// TIA Portal V20 export
FUNCTION_BLOCK "Simulation"   // FB193, LAD
// stored: MemoryReserve 100, Namespace Unit1.Em4, SetENOAutomatically false
   VAR_INPUT
      simulation { ExternalAccessible := 'False'; ExternalVisible := 'False'; ExternalWritable := 'False'} : Bool;
   END_VAR
   VAR
      instActuator { ExternalAccessible := 'False'; ExternalVisible := 'False'; ExternalWritable := 'False'} : Array[0..19] of "Simulation_Actuator";
      statDigitalSignal { ExternalAccessible := 'False'; ExternalVisible := 'False'; ExternalWritable := 'False'} : Array[0..9] of Bool;
   END_VAR
   VAR_TEMP
      tempTRPnPleftPlace : Bool;
   END_VAR
   VAR_TEMP   // added for the SCL form of the ladder/FBD networks
      _w1 : Bool;
   END_VAR
BEGIN

REGION Network 1: Digital Signal
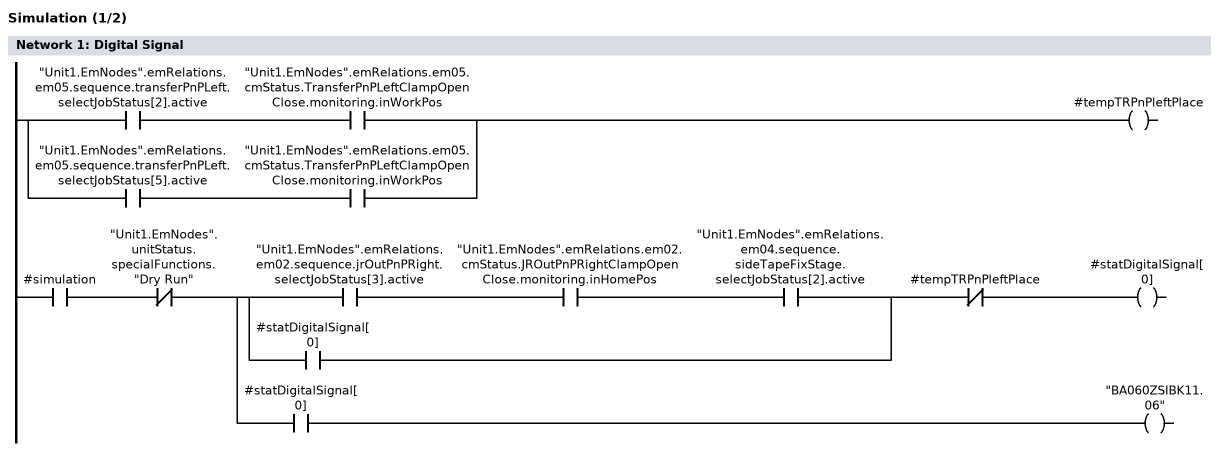
   RUNG wire#powerrail
      Contact( "Unit1.EmNodes".emRelations.em05.sequence.transferPnPLeft.selectJobStatus[2].active )
      Contact( "Unit1.EmNodes".emRelations.em05.cmStatus.TransferPnPLeftClampOpenClose.monitoring.inWorkPos )
      wire#w1
      Coil( #tempTRPnPleftPlace )
   END_RUNG
   RUNG wire#powerrail
      Contact( "Unit1.EmNodes".emRelations.em05.sequence.transferPnPLeft.selectJobStatus[5].active )
      Contact( "Unit1.EmNodes".emRelations.em05.cmStatus.TransferPnPLeftClampOpenClose.monitoring.inWorkPos )
   END_RUNG wire#w1
   RUNG wire#powerrail
      Contact( #simulation )
      I_Contact( "Unit1.EmNodes".unitStatus.specialFunctions."Dry Run" )
      wire#w2
      Contact( "Unit1.EmNodes".emRelations.em02.sequence.jrOutPnPRight.selectJobStatus[3].active )
      Contact( "Unit1.EmNodes".emRelations.em02.cmStatus.JROutPnPRightClampOpenClose.monitoring.inHomePos )
      Contact( "Unit1.EmNodes".emRelations.em04.sequence.sideTapeFixStage.selectJobStatus[2].active )
      wire#w3
      I_Contact( #tempTRPnPleftPlace )
      Coil( #statDigitalSignal[0] )
   END_RUNG
   RUNG wire#w2
      Contact( #statDigitalSignal[0] )
   END_RUNG wire#w3
   RUNG wire#w2
      Contact( #statDigitalSignal[0] )
      Coil( "BA060ZSIBK11.06" )
   END_RUNG
   // the same network as SCL:
   #tempTRPnPleftPlace := ("Unit1.EmNodes".emRelations.em05.sequence.transferPnPLeft.selectJobStatus[2].active AND "Unit1.EmNodes".emRelations.em05.cmStatus.TransferPnPLeftClampOpenClose.monitoring.inWorkPos) OR ("Unit1.EmNodes".emRelations.em05.sequence.transferPnPLeft.selectJobStatus[5].active AND "Unit1.EmNodes".emRelations.em05.cmStatus.TransferPnPLeftClampOpenClose.monitoring.inWorkPos);
   #_w1 := #simulation AND NOT "Unit1.EmNodes".unitStatus.specialFunctions."Dry Run";
   #statDigitalSignal[0] := #_w1 AND (("Unit1.EmNodes".emRelations.em02.sequence.jrOutPnPRight.selectJobStatus[3].active AND "Unit1.EmNodes".emRelations.em02.cmStatus.JROutPnPRightClampOpenClose.monitoring.inHomePos AND "Unit1.EmNodes".emRelations.em04.sequence.sideTapeFixStage.selectJobStatus[2].active) OR #statDigitalSignal[0]) AND NOT #tempTRPnPleftPlace;
   "BA060ZSIBK11.06" := #_w1 AND #statDigitalSignal[0];
END_REGION

REGION Network 2: Two Way Actuator
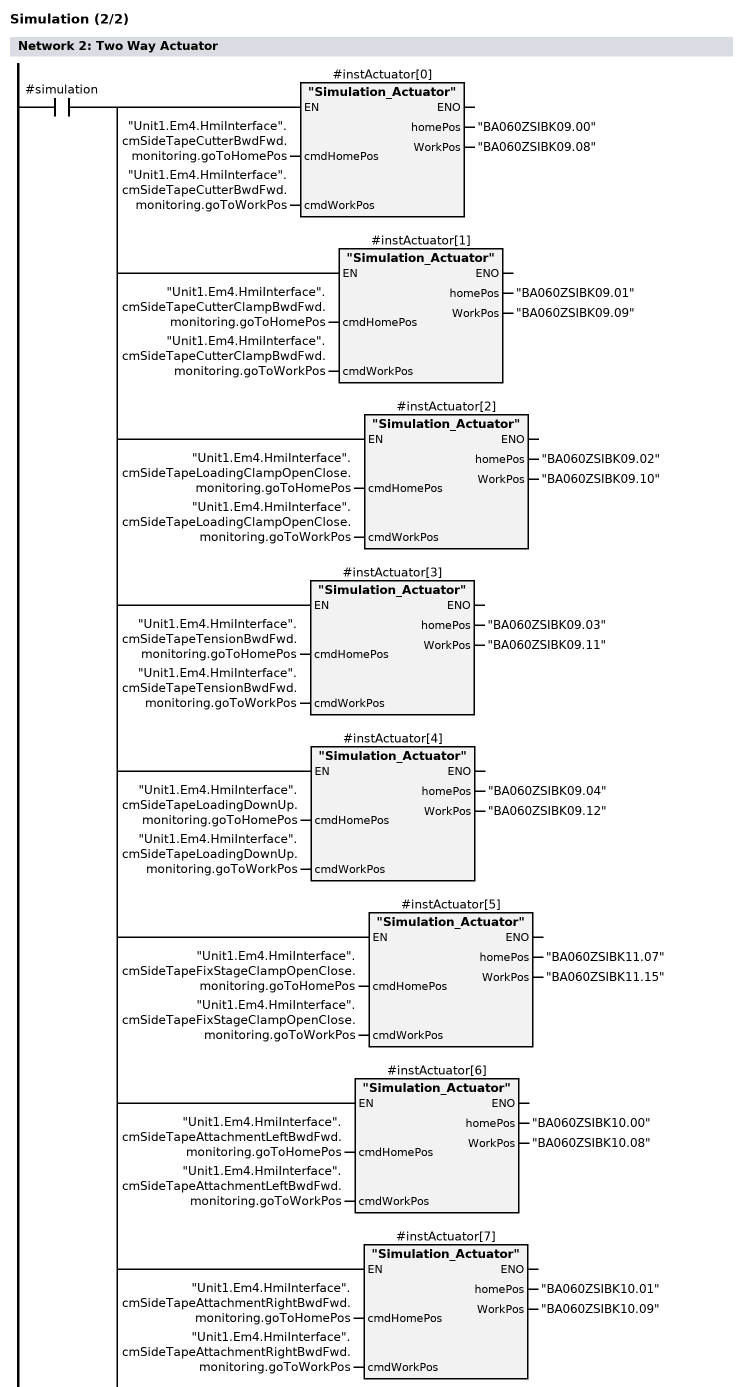
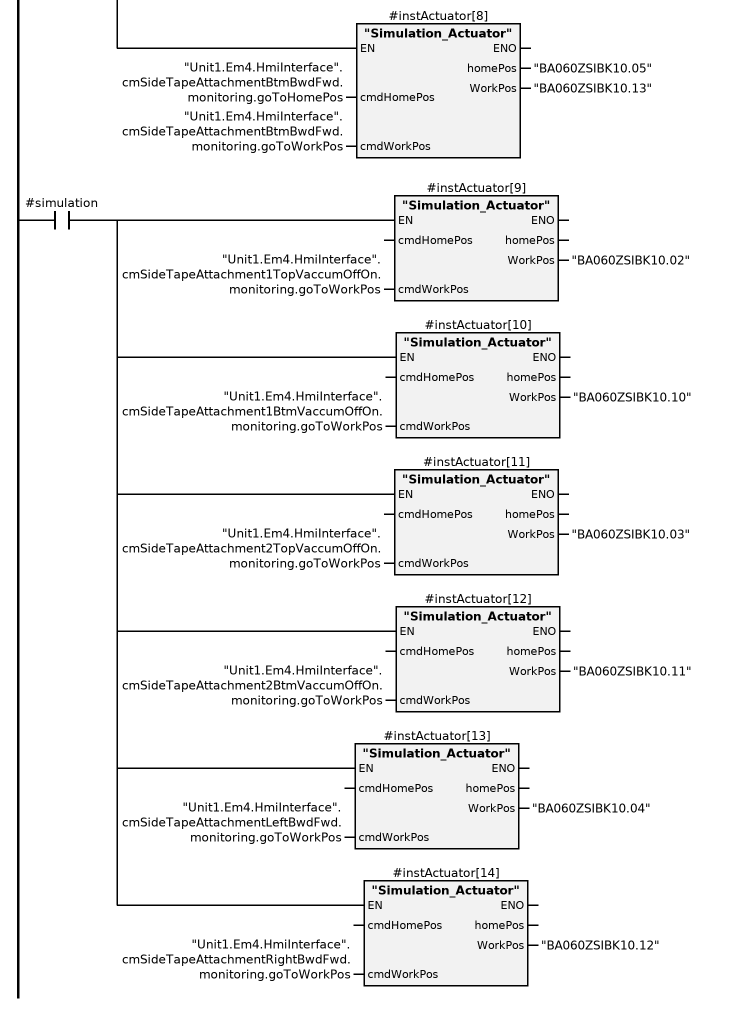
   RUNG wire#powerrail
      Contact( #simulation )
      wire#w1
      #instActuator[0](cmdHomePos := "Unit1.Em4.HmiInterface".cmSideTapeCutterBwdFwd.monitoring.goToHomePos, cmdWorkPos := "Unit1.Em4.HmiInterface".cmSideTapeCutterBwdFwd.monitoring.goToWorkPos, homePos => "BA060ZSIBK09.00", WorkPos => "BA060ZSIBK09.08")
   END_RUNG
   RUNG wire#w1
      #instActuator[1](cmdHomePos := "Unit1.Em4.HmiInterface".cmSideTapeCutterClampBwdFwd.monitoring.goToHomePos, cmdWorkPos := "Unit1.Em4.HmiInterface".cmSideTapeCutterClampBwdFwd.monitoring.goToWorkPos, homePos => "BA060ZSIBK09.01", WorkPos => "BA060ZSIBK09.09")
   END_RUNG
   RUNG wire#w1
      #instActuator[2](cmdHomePos := "Unit1.Em4.HmiInterface".cmSideTapeLoadingClampOpenClose.monitoring.goToHomePos, cmdWorkPos := "Unit1.Em4.HmiInterface".cmSideTapeLoadingClampOpenClose.monitoring.goToWorkPos, homePos => "BA060ZSIBK09.02", WorkPos => "BA060ZSIBK09.10")
   END_RUNG
   RUNG wire#w1
      #instActuator[3](cmdHomePos := "Unit1.Em4.HmiInterface".cmSideTapeTensionBwdFwd.monitoring.goToHomePos, cmdWorkPos := "Unit1.Em4.HmiInterface".cmSideTapeTensionBwdFwd.monitoring.goToWorkPos, homePos => "BA060ZSIBK09.03", WorkPos => "BA060ZSIBK09.11")
   END_RUNG
   RUNG wire#w1
      #instActuator[4](cmdHomePos := "Unit1.Em4.HmiInterface".cmSideTapeLoadingDownUp.monitoring.goToHomePos, cmdWorkPos := "Unit1.Em4.HmiInterface".cmSideTapeLoadingDownUp.monitoring.goToWorkPos, homePos => "BA060ZSIBK09.04", WorkPos => "BA060ZSIBK09.12")
   END_RUNG
   RUNG wire#w1
      #instActuator[5](cmdHomePos := "Unit1.Em4.HmiInterface".cmSideTapeFixStageClampOpenClose.monitoring.goToHomePos, cmdWorkPos := "Unit1.Em4.HmiInterface".cmSideTapeFixStageClampOpenClose.monitoring.goToWorkPos, homePos => "BA060ZSIBK11.07", WorkPos => "BA060ZSIBK11.15")
   END_RUNG
   RUNG wire#w1
      #instActuator[6](cmdHomePos := "Unit1.Em4.HmiInterface".cmSideTapeAttachmentLeftBwdFwd.monitoring.goToHomePos, cmdWorkPos := "Unit1.Em4.HmiInterface".cmSideTapeAttachmentLeftBwdFwd.monitoring.goToWorkPos, homePos => "BA060ZSIBK10.00", WorkPos => "BA060ZSIBK10.08")
   END_RUNG
   RUNG wire#w1
      #instActuator[7](cmdHomePos := "Unit1.Em4.HmiInterface".cmSideTapeAttachmentRightBwdFwd.monitoring.goToHomePos, cmdWorkPos := "Unit1.Em4.HmiInterface".cmSideTapeAttachmentRightBwdFwd.monitoring.goToWorkPos, homePos => "BA060ZSIBK10.01", WorkPos => "BA060ZSIBK10.09")
   END_RUNG
   RUNG wire#w1
      #instActuator[8](cmdHomePos := "Unit1.Em4.HmiInterface".cmSideTapeAttachmentBtmBwdFwd.monitoring.goToHomePos, cmdWorkPos := "Unit1.Em4.HmiInterface".cmSideTapeAttachmentBtmBwdFwd.monitoring.goToWorkPos, homePos => "BA060ZSIBK10.05", WorkPos => "BA060ZSIBK10.13")
   END_RUNG
   RUNG wire#powerrail
      Contact( #simulation )
      wire#w2
      #instActuator[9](cmdHomePos :=, cmdWorkPos := "Unit1.Em4.HmiInterface".cmSideTapeAttachment1TopVaccumOffOn.monitoring.goToWorkPos, homePos =>, WorkPos => "BA060ZSIBK10.02")
   END_RUNG
   RUNG wire#w2
      #instActuator[10](cmdHomePos :=, cmdWorkPos := "Unit1.Em4.HmiInterface".cmSideTapeAttachment1BtmVaccumOffOn.monitoring.goToWorkPos, homePos =>, WorkPos => "BA060ZSIBK10.10")
   END_RUNG
   RUNG wire#w2
      #instActuator[11](cmdHomePos :=, cmdWorkPos := "Unit1.Em4.HmiInterface".cmSideTapeAttachment2TopVaccumOffOn.monitoring.goToWorkPos, homePos =>, WorkPos => "BA060ZSIBK10.03")
   END_RUNG
   RUNG wire#w2
      #instActuator[12](cmdHomePos :=, cmdWorkPos := "Unit1.Em4.HmiInterface".cmSideTapeAttachment2BtmVaccumOffOn.monitoring.goToWorkPos, homePos =>, WorkPos => "BA060ZSIBK10.11")
   END_RUNG
   RUNG wire#w2
      #instActuator[13](cmdHomePos :=, cmdWorkPos := "Unit1.Em4.HmiInterface".cmSideTapeAttachmentLeftBwdFwd.monitoring.goToWorkPos, homePos =>, WorkPos => "BA060ZSIBK10.04")
   END_RUNG
   RUNG wire#w2
      #instActuator[14](cmdHomePos :=, cmdWorkPos := "Unit1.Em4.HmiInterface".cmSideTapeAttachmentRightBwdFwd.monitoring.goToWorkPos, homePos =>, WorkPos => "BA060ZSIBK10.12")
   END_RUNG
   // the same network as SCL:
   IF #simulation THEN
       #instActuator[0](cmdHomePos := "Unit1.Em4.HmiInterface".cmSideTapeCutterBwdFwd.monitoring.goToHomePos,   // "Simulation_Actuator"
                        cmdWorkPos := "Unit1.Em4.HmiInterface".cmSideTapeCutterBwdFwd.monitoring.goToWorkPos,
                        homePos => "BA060ZSIBK09.00",
                        WorkPos => "BA060ZSIBK09.08");
       #instActuator[1](cmdHomePos := "Unit1.Em4.HmiInterface".cmSideTapeCutterClampBwdFwd.monitoring.goToHomePos,   // "Simulation_Actuator"
                        cmdWorkPos := "Unit1.Em4.HmiInterface".cmSideTapeCutterClampBwdFwd.monitoring.goToWorkPos,
                        homePos => "BA060ZSIBK09.01",
                        WorkPos => "BA060ZSIBK09.09");
       #instActuator[2](cmdHomePos := "Unit1.Em4.HmiInterface".cmSideTapeLoadingClampOpenClose.monitoring.goToHomePos,   // "Simulation_Actuator"
                        cmdWorkPos := "Unit1.Em4.HmiInterface".cmSideTapeLoadingClampOpenClose.monitoring.goToWorkPos,
                        homePos => "BA060ZSIBK09.02",
                        WorkPos => "BA060ZSIBK09.10");
       #instActuator[3](cmdHomePos := "Unit1.Em4.HmiInterface".cmSideTapeTensionBwdFwd.monitoring.goToHomePos,   // "Simulation_Actuator"
                        cmdWorkPos := "Unit1.Em4.HmiInterface".cmSideTapeTensionBwdFwd.monitoring.goToWorkPos,
                        homePos => "BA060ZSIBK09.03",
                        WorkPos => "BA060ZSIBK09.11");
       #instActuator[4](cmdHomePos := "Unit1.Em4.HmiInterface".cmSideTapeLoadingDownUp.monitoring.goToHomePos,   // "Simulation_Actuator"
                        cmdWorkPos := "Unit1.Em4.HmiInterface".cmSideTapeLoadingDownUp.monitoring.goToWorkPos,
                        homePos => "BA060ZSIBK09.04",
                        WorkPos => "BA060ZSIBK09.12");
       #instActuator[5](cmdHomePos := "Unit1.Em4.HmiInterface".cmSideTapeFixStageClampOpenClose.monitoring.goToHomePos,   // "Simulation_Actuator"
                        cmdWorkPos := "Unit1.Em4.HmiInterface".cmSideTapeFixStageClampOpenClose.monitoring.goToWorkPos,
                        homePos => "BA060ZSIBK11.07",
                        WorkPos => "BA060ZSIBK11.15");
       #instActuator[6](cmdHomePos := "Unit1.Em4.HmiInterface".cmSideTapeAttachmentLeftBwdFwd.monitoring.goToHomePos,   // "Simulation_Actuator"
                        cmdWorkPos := "Unit1.Em4.HmiInterface".cmSideTapeAttachmentLeftBwdFwd.monitoring.goToWorkPos,
                        homePos => "BA060ZSIBK10.00",
                        WorkPos => "BA060ZSIBK10.08");
       #instActuator[7](cmdHomePos := "Unit1.Em4.HmiInterface".cmSideTapeAttachmentRightBwdFwd.monitoring.goToHomePos,   // "Simulation_Actuator"
                        cmdWorkPos := "Unit1.Em4.HmiInterface".cmSideTapeAttachmentRightBwdFwd.monitoring.goToWorkPos,
                        homePos => "BA060ZSIBK10.01",
                        WorkPos => "BA060ZSIBK10.09");
       #instActuator[8](cmdHomePos := "Unit1.Em4.HmiInterface".cmSideTapeAttachmentBtmBwdFwd.monitoring.goToHomePos,   // "Simulation_Actuator"
                        cmdWorkPos := "Unit1.Em4.HmiInterface".cmSideTapeAttachmentBtmBwdFwd.monitoring.goToWorkPos,
                        homePos => "BA060ZSIBK10.05",
                        WorkPos => "BA060ZSIBK10.13");
       #instActuator[9](cmdWorkPos := "Unit1.Em4.HmiInterface".cmSideTapeAttachment1TopVaccumOffOn.monitoring.goToWorkPos,   // "Simulation_Actuator"
                        WorkPos => "BA060ZSIBK10.02");
       #instActuator[10](cmdWorkPos := "Unit1.Em4.HmiInterface".cmSideTapeAttachment1BtmVaccumOffOn.monitoring.goToWorkPos,   // "Simulation_Actuator"
                         WorkPos => "BA060ZSIBK10.10");
       #instActuator[11](cmdWorkPos := "Unit1.Em4.HmiInterface".cmSideTapeAttachment2TopVaccumOffOn.monitoring.goToWorkPos,   // "Simulation_Actuator"
                         WorkPos => "BA060ZSIBK10.03");
       #instActuator[12](cmdWorkPos := "Unit1.Em4.HmiInterface".cmSideTapeAttachment2BtmVaccumOffOn.monitoring.goToWorkPos,   // "Simulation_Actuator"
                         WorkPos => "BA060ZSIBK10.11");
       #instActuator[13](cmdWorkPos := "Unit1.Em4.HmiInterface".cmSideTapeAttachmentLeftBwdFwd.monitoring.goToWorkPos,   // "Simulation_Actuator"
                         WorkPos => "BA060ZSIBK10.04");
       #instActuator[14](cmdWorkPos := "Unit1.Em4.HmiInterface".cmSideTapeAttachmentRightBwdFwd.monitoring.goToWorkPos,   // "Simulation_Actuator"
                         WorkPos => "BA060ZSIBK10.12");
   END_IF;
END_REGION

REGION Network 3 (SCL): homing
   IF #simulation AND "JB_Temp".Test_Homing[4] THEN

       "Unit1.Em4.HmiInterface".cmSideTapeFixStageAxisX.commands.homing :=
       "Unit1.Em4.HmiInterface".cmSideTapeFixStageAxisC.commands.homing :=
       "Unit1.Em4.HmiInterface".cmSideTapeAttachmentAxisX.commands.homing :=
       "Unit1.Em4.HmiInterface".cmSideTapeAttachmentAxisY.commands.homing := true;

       "Unit1.Em4.HmiInterface".cmSideTapeAttachment1TopVaccumOffOn.commands.commandHomePos :=
       "Unit1.Em4.HmiInterface".cmSideTapeAttachment1BtmVaccumOffOn.commands.commandHomePos :=
       "Unit1.Em4.HmiInterface".cmSideTapeAttachment2TopVaccumOffOn.commands.commandHomePos :=
       "Unit1.Em4.HmiInterface".cmSideTapeAttachment2BtmVaccumOffOn.commands.commandHomePos :=
       "Unit1.Em4.HmiInterface".cmSideTapeAttachmentLeftBwdFwd.commands.commandHomePos :=
       "Unit1.Em4.HmiInterface".cmSideTapeAttachmentRightBwdFwd.commands.commandHomePos :=
       "Unit1.Em4.HmiInterface".cmSideTapeAttachmentBtmBwdFwd.commands.commandWorkPos :=
       "Unit1.Em4.HmiInterface".cmSideTapeLoadingClampOpenClose.commands."commandHomePos" := true;

       "JB_Temp".Test_Homing[4] := false;
   //    
   END_IF;

   IF #simulation AND "JB_Temp".Test_Homing[20] THEN


       "Unit1.Em4.HmiInterface".cmSideTapeFixStageAxisX.commands.homing :=
       "Unit1.Em4.HmiInterface".cmSideTapeFixStageAxisC.commands.homing :=
       "Unit1.Em4.HmiInterface".cmSideTapeAttachmentAxisX.commands.homing :=
       "Unit1.Em4.HmiInterface".cmSideTapeAttachmentAxisY.commands.homing :=

       "Unit1.Em4.HmiInterface".cmSideTapeAttachment2TopVaccumOffOn.commands.commandHomePos :=
       "Unit1.Em4.HmiInterface".cmSideTapeAttachment2BtmVaccumOffOn.commands.commandHomePos :=
       "Unit1.Em4.HmiInterface".cmSideTapeAttachmentLeftBwdFwd.commands.commandHomePos :=
       "Unit1.Em4.HmiInterface".cmSideTapeAttachmentRightBwdFwd.commands.commandHomePos :=
       "Unit1.Em4.HmiInterface".cmSideTapeAttachmentBtmBwdFwd.commands.commandWorkPos :=
       "Unit1.Em4.HmiInterface".cmSideTapeLoadingClampOpenClose.commands."commandHomePos" := false;
   END_IF;
END_REGION
END_FUNCTION_BLOCK
